(*
SPDX-FileCopyrightText: © 2026 Oleksandr Tiutyk <trofimich@gmail.com>
SPDX-License-Identifier: MIT
License: https://opensource.org/license/mit
*)

(*!
<summary>Owns the namespace storage shared by FileSystem diagnostic metadata.</summary>
*)

{attribute 'no_explicit_call' := 'do not call this POU directly'}
PROGRAM INTERNAL CurrentNamespace
VAR
	{attribute 'hide'} 
	_NamespaceExtractor : NamespaceExtractor;
END_VAR

(*!
<summary>Provides the compiler-initialized namespace string for this library.</summary>
<description>Returns borrowed read-only storage owned by the internal namespace extractor.</description>
*)
{attribute 'monitoring' := 'call'}
PROPERTY Name : REFERENCE TO STRING
GET
Name REF= _NamespaceExtractor.CurrentNamespace;
END_GET
END_PROPERTY

END_PROGRAM

(* stored: Version 1.1.0.1
   POU CurrentNamespace: Id {f24d7c34-d6e3-45a4-9a69-d0c668832c17}, SpecialFunc None
   Property Name: Id {ab92da57-5dc1-4458-91d8-c6f305012951}
   Get Get: Id {768d7488-7081-4761-adfb-5b76040ddcb9} *)
